FUNCTION_BLOCK Piper_Test EXTENDS FB_TestSuite
VAR_INPUT
END_VAR
VAR_OUTPUT
END_VAR
VAR
END_VAR

// Copyright (c) 2024 Loupe (https://loupe.team), provided under the MIT License.

CommandSetsState();
StateTransitions();

METHOD AbortAndClear
VAR_INPUT
    piper : REFERENCE TO Piper;
END_VAR
// Copyright (c) 2024 Loupe (https://loupe.team), provided under the MIT License.

piper.command.Abort := TRUE;
piper();
AssertEquals_DINT(piper.packMLState, MACHINE_STATE.ABORTING, Message := 'State should be ABORTING');
piper.NextState();
AssertEquals_DINT(piper.packMLState, MACHINE_STATE.ABORTED, Message := 'State after STARTING should be ABORTED');

piper.command.Clear := TRUE;
piper();
AssertEquals_DINT(piper.packMLState, MACHINE_STATE.CLEARING, Message := 'State should be CLEARING');
piper.NextState();
AssertEquals_DINT(piper.packMLState, MACHINE_STATE.STOPPED, Message := 'State after CLEARING should be STOPPED');
END_METHOD

METHOD CommandSetsState
VAR
    piper : Piper;
END_VAR
// Copyright (c) 2024 Loupe (https://loupe.team), provided under the MIT License.

// Check that state actually gets set
// Run this sanity check before the full state transition checks
TEST('SetState');
piper.command.Reset := TRUE;
piper();
AssertFalse(piper.command.Reset, Message := 'Command should be cyclicly reset');
AssertEquals_DINT(piper.packMLState,
    MACHINE_STATE.RESETTING,
    Message := 'Setting a valid state command and cyclic calling FUB once should change state');

TEST_FINISHED();
END_METHOD

METHOD Holding : BOOL
VAR_INPUT
    piper : REFERENCE TO Piper;
END_VAR
// Copyright (c) 2024 Loupe (https://loupe.team), provided under the MIT License.

piper.command.Hold := TRUE;
piper();
AssertEquals_DINT(Expected := piper.packMLState, Actual := MACHINE_STATE.HOLDING, Message := 'State should be HOLDING');
END_METHOD

METHOD Resetting
VAR_INPUT
    piper : REFERENCE TO Piper;
END_VAR
// Copyright (c) 2024 Loupe (https://loupe.team), provided under the MIT License.

piper.command.Reset := TRUE;
piper();
AssertEquals_DINT(Expected := piper.packMLState, Actual := MACHINE_STATE.RESETTING, Message := 'State should be RESETTING');
END_METHOD

METHOD StartAndExecute : BOOL
VAR_INPUT
    piper : REFERENCE TO Piper;
END_VAR
// Copyright (c) 2024 Loupe (https://loupe.team), provided under the MIT License.

piper.command.Start := TRUE;
piper();
AssertEquals_DINT(piper.packMLState, MACHINE_STATE.STARTING, Message := 'State should be STARTING');
piper.NextState();
piper();
END_METHOD

METHOD Starting
VAR_INPUT
    piper : REFERENCE TO Piper;
END_VAR
// Copyright (c) 2024 Loupe (https://loupe.team), provided under the MIT License.

piper.command.Start := TRUE;
piper();
AssertEquals_DINT(piper.packMLState, MACHINE_STATE.STARTING, Message := 'State should be STARTING');
END_METHOD

METHOD StateTransitions
VAR
    piper : Piper();
    task : TaskFB();
    piperModule : Piper_EM(piper, task);
END_VAR
// Copyright (c) 2024 Loupe (https://loupe.team), provided under the MIT License.

// This test confirms the order of state progressions per PackML (with additional BOOTING state)
// With no submodules, it's expected Piper will proceed immediately to the next state

(*STweep.Disable*)

TEST('BootAndReset');
	// Note: there is currently no abort while booting
	AssertEquals_DINT(piper.packMLState, MACHINE_STATE.BOOTING, Message := 'Initil state should be BOOTING');
	piper.NextState();
	AssertEquals_DINT(piper.packMLState, MACHINE_STATE.STOPPED, Message := 'STOPPED state should be after BOOTING');
	
	Resetting(piper);
	piper.NextState();
	AssertEquals_DINT(piper.packMLState, MACHINE_STATE.IDLE, Message := 'Next state after RESETTING should be IDLE');

TEST_FINISHED();

TEST('StartAndAbortWhileStarting');
	Starting(piper);
	
	AbortAndClear(piper);
	
	Resetting(piper);
	piper.NextState();
	AssertEquals_DINT(piper.packMLState, MACHINE_STATE.IDLE, Message := 'Next state after RESETTING should be IDLE');
TEST_FINISHED();

TEST('ResetAndAbortWhileResetting');
	AbortAndClear(piper); // Get into CLEARED
	Resetting(piper);
	// in resetting
	AbortAndClear(piper);
	// stopped
	Resetting(piper);
	piper.NextState();
	AssertEquals_DINT(piper.packMLState, MACHINE_STATE.IDLE, Message := 'Next state after RESETTING should be IDLE');
TEST_FINISHED();

TEST('ExecuteAndAbortWhileExecuting');
	Starting(piper);
	piper.NextState(); // in Executing
	AbortAndClear(piper);
	// stopped
	Resetting(piper);
	piper.NextState();
	AssertEquals_DINT(piper.packMLState, MACHINE_STATE.IDLE, Message := 'Next state after RESETTING should be IDLE');
TEST_FINISHED();

TEST('ExecuteAndStop');
	Starting(piper);
	piper.NextState(); // in Executing
	
	Stopping(piper);
	piper.NextState();
	// stopped
	Resetting(piper);
	piper.NextState();
	AssertEquals_DINT(piper.packMLState, MACHINE_STATE.IDLE, Message := 'Next state after RESETTING should be IDLE');
TEST_FINISHED();

//TEST('HoldAndUnhold');
//	piper.RegisterSubmodule(piperModule);
//	Starting(piper);
//	piper.NextState(); // in Executing

//	Holding(piper);
//	Unholding(piper);

//	Stopping(piper);
//	piper.NextState();
//	// stopped
//	Resetting(piper);
//	piper.NextState();
//	AssertEquals_DINT(piper.PackMLState, MACHINE_STATE.IDLE, Message := 'Next state after RESETTING should be IDLE');
//TEST_FINISHED();

//TEST('SuspendAndUnSuspend');
//	Starting(piper);
//	piper.NextState(); // in Executing

//	Suspending(piper);
//	Unsuspending(piper);

//	Stopping(piper);
//	piper.NextState();
//	// stopped
//	Resetting(piper);
//	piper.NextState();
//	AssertEquals_DINT(piper.PackMLState, MACHINE_STATE.IDLE, Message := 'Next state after RESETTING should be IDLE');
//TEST_FINISHED();
END_METHOD

METHOD Stopping : BOOL
VAR_INPUT
    piper : REFERENCE TO Piper;
END_VAR
// Copyright (c) 2024 Loupe (https://loupe.team), provided under the MIT License.

piper.command.Stop := TRUE;
piper();
AssertEquals_DINT(piper.packMLState, MACHINE_STATE.STOPPING, Message := 'State should be STOPPING');
END_METHOD

METHOD Suspending : BOOL
VAR_INPUT
    piper : REFERENCE TO Piper;
END_VAR
// Copyright (c) 2024 Loupe (https://loupe.team), provided under the MIT License.

piper.command.Suspend := TRUE;
piper();
AssertEquals_DINT(Expected := piper.packMLState, Actual := MACHINE_STATE.SUSPENDING, Message := 'State should be SUSPENDING');
END_METHOD

METHOD Unholding : BOOL
VAR_INPUT
    piper : REFERENCE TO Piper;
END_VAR
// Copyright (c) 2024 Loupe (https://loupe.team), provided under the MIT License.

piper.command.Unhold := TRUE;
piper();
AssertEquals_DINT(Expected := piper.packMLState, Actual := MACHINE_STATE.UNHOLDING, Message := 'State should be UNHOLDING');
END_METHOD

METHOD Unsuspending : BOOL
VAR_INPUT
    piper : REFERENCE TO Piper;
END_VAR
// Copyright (c) 2024 Loupe (https://loupe.team), provided under the MIT License.

piper.command.Unsuspend := TRUE;
piper();
AssertEquals_DINT(Expected := piper.packMLState, Actual := MACHINE_STATE.UNSUSPENDING, Message := 'State should be UNSUSPENDING');
END_METHOD

END_FUNCTION_BLOCK

(* stored: Version 1.1.0.1
   POU Piper_Test: Id {68fc7220-a76f-05fc-0e18-f4d46c3c0059}, SpecialFunc None
   Folder PartialTestsForStateTransitions: Id {02880b83-610a-097b-2248-8bc540cec99f}
   Method AbortAndClear: Id {c5c2e356-af92-0470-06c7-0552a5a2869e}
   Method CommandSetsState: Id {c0302bd5-f07a-06ee-1d5c-15fc195e6380}
   Method Holding: Id {1ccbe795-9e71-0deb-2652-90d9a7429477}
   Method Resetting: Id {442f8c1d-3e24-0484-05f8-c450bb57964e}
   Method StartAndExecute: Id {1503700b-a107-092d-0dda-dabd453b3226}
   Method Starting: Id {1a40e8b9-782b-0c9e-1434-1b3a5144a2db}
   Method StateTransitions: Id {0bcdaa3a-ee87-022d-33ad-b2aa61c63cc5}
   Method Stopping: Id {674f0d8d-b58f-0301-35f4-696c54818e38}
   Method Suspending: Id {0729cdc7-2784-0ac8-0f52-122ac02f1e89}
   Method Unholding: Id {2edea14a-06a7-0455-011d-6b1dd451c7c5}
   Method Unsuspending: Id {9f5295b8-2127-095f-05f0-00362851360a} *)
